Universal Robots PolyScope program: Cobot_soudure_29112023.urp

Program Cobot_soudure_29112023 (installation=Cobot_soudure_29112023 directory=/home/ur/ursim/ursim-5.11.0.108249/programs/TRAVAIL 27112023 createdIn=5.9.4.1031232 lastSavedIn=5.11.0.108249 robotSerialNumber=20195299999)
Calibrated DH parameters: a=[0, -0.6127, -0.57155, 0, 0, 0]; d=[0.1807, 0, 0, 0.17415, 0.11985, 0.11655]; alpha=[1.570796, 0, 0, 1.570796, -1.570796, 0]; deltaTheta=[0, 0, 0, 0, 0, 0]
InitVariablesNode variables(variable(name=Test_Gaz, expression=False), variable(name=Test_Job, expression=False), variable(name=Test_Ordre_Mar, expression=False), variable(name=Valide_Gaz, expression=False), variable(name=fin_soud, expression=1), variable(name=secu_d, expression=0), variable(name=secu_g, expression=0), variable(name=timer_ret_gaz, expression=0))
BeforeStart
  Folder fonctions
    Folder Init [hidden by the author, left out]
    Folder Diverses
      Script file /home/ur/ursim/ursim-5.11.0.108249/programs/SCRIPT/Scripts_soudure/Diverses/close_popup.script
        | #fermeture popup
        | 
        | def close_popup():
        | 	closepop = "close popup"
        |     	socket_send_string(closepop,"internal")
        |     	socket_send_byte(10,"internal")
        |     	socket_close()
        | 
        | 	closepop = "close popup"
        |     	socket_send_string(closepop,"internal")
        |     	socket_send_byte(10,"internal")
        |     	socket_close()
        | 	return(False)
        | end
      Script file /home/ur/ursim/ursim-5.11.0.108249/programs/SCRIPT/Scripts_soudure/Diverses/debut_soud.script
        | def fun_debut_soudure():
        |     Valide_Gaz = False
        |     if  ((Test_Ordre_Mar == False) and (Test_Job == False)):
        |         Arc_On = True
        |         Test_Gaz = True
        |     end
        | end
      Script file /home/ur/ursim/ursim-5.11.0.108249/programs/SCRIPT/Scripts_soudure/Diverses/fin_soudure.script
        | def fin_soudure():
        |         Arc_On = False
        |         Test_Gaz = False
        |         Test_Job = True
        |         Test_Ordre_Mar = True
        | end
      Script file /home/ur/ursim/ursim-5.11.0.108249/programs/SCRIPT/Scripts_soudure/Diverses/fun_demande_job.script
        | #demande le job à utiliser (mode de soudure régler sur le poste à souder) (compris entre 0 et 3, pour 1 et 4 sur le poste a souder)
        | def fun_demande_job(type):
        | 	if (1==type):
        | 		soudure = "point"
        | 	elif (2==type):
        | 		soudure = "lineaire"
        | 	elif (3==type):
        | 		soudure = "arc de cercle"
        | 	elif (4==type):
        | 		soudure = "cercle"
        | 	elif (5==type):
        | 		soudure = "lineaire + balayage"
        | 	elif (6==type):
        | 		soudure = "Recopie"
        | 	else :
        | 		return(False)
        | 	end
        | 
        |   job = request_integer_from_primary_client("Mode du poste à souder pour soudure : "+ soudure + " ? [1-4]")
        |   #job = job-1 #adapter la saisie aux besoins du code
        | 
        |   while ((job!=4) and (job!=1) and (job!=2) and (job!=3)): #reboucler si mauvaise saisie
        | 	  job = request_integer_from_primary_client("Mode du poste à souder pour soudure : "+ soudure + " ? [1-4]")
        |       #job = job-1 #adapter la saisie aux besoins du code
        |   end
        | 
        | return(job)
        | end
      Script file /home/ur/ursim/ursim-5.11.0.108249/programs/SCRIPT/Scripts_soudure/Diverses/fun_demande_type_soudure.script
        | #demande le type de soudure à enregistrer (entre 1 et 5)
        | def fun_demande_type_soudure():
        |     sync()
        | 	reponse = request_integer_from_primary_client("1->POINT     2->LINEAIRE    3->ARC    4->CERCLE  5->LINEAIRE BALAYAGE     6->RECOPIE     7->FIN")
        |     sync()
        |     if ((reponse == 0) or (reponse >= 7)):
        |         reponse = 7
        |     end
        |     sync()
        | return(reponse)
        | end
      SuppressedNode
        Script file /home/ur/ursim/ursim-5.11.0.108249/programs/SCRIPT/Scripts_soudure/Diverses/fun_demande().script
          | #demande nombre soudures par type (compris entre 0 et 6)
          | 
          | def fun_demande(type):
          | 	if (1==type):
          | 		soudure = "point"					#si type = 1, la demande sera sur une soudure point
          | 	elif (2==type):
          | 		soudure = "lineaire"				#si type = 2, la demande sera sur une soudure linéaire
          | 	elif (3==type):
          | 		soudure = "arc de cercle"			#si type = 3, la demande sera sur une soudure arc de cercle
          | 	elif (4==type):
          | 		soudure = "cercle"					#si type = 4, la demande sera sur une soudure cercle
          | 	elif (5==type):
          | 		soudure = "lineaire + balayage"
          | 	else :
          | 		return(False)
          | 	end
          | 
          | 	nb_soud = request_integer_from_primary_client("nombre de soudure(s) "+ soudure + " ?")			#la demande
          | 	if (nb_soud >6):																									#si la reponse est superieur a 6
          | 		popup1 = "popup le robot ne peut pas effectuer plus de 6 soudures "+ soudure + " sur la même pièce, réessayer."	#popup
          | 		socket_open("127.0.0.1",29999,"internal") # open internal socket
          | 
          | 		socket_send_line(popup1,"internal")         #Affichage Popup
          | 
          | 		socket_send_byte(10,"internal")
          | 		sleep(5.0)
          | 		closepop = "close popup"					#fermer popup
          | 		socket_send_string(closepop,"internal")
          | 		socket_send_byte(10,"internal")
          | 		socket_close()
          | 
          | 		while(nb_soud >6):
          | 			nb_soud = request_integer_from_primary_client("nombre de soudure(s) "+ soudure + " ? (compris entre 0 et 6 ;)")	#on redemande tant que le nombre est superieur a 6
          | 		end
          | end
          | return(nb_soud)        #on retourne le nombre de soudure à effectuer dans le type
          | end
      Script file /home/ur/ursim/ursim-5.11.0.108249/programs/SCRIPT/Scripts_soudure/Diverses/fun_demande_vit.script
        | #demande nombre soudures par type (compris entre 0 et 6)
        | def fun_demande_vit(type):
        | 	if (1==type):
        | 		soudure = "point"
        | 	elif (2==type):
        | 		soudure = "lineaire"
        | 	elif (3==type):
        | 		soudure = "arc de cercle"
        | 	elif (4==type):
        | 		soudure = "cercle"
        | 	else :
        | 		return(False)
        | 	end
        | 
        | vit_soud = request_float_from_primary_client("vitesse de la soudure "+ soudure + " ? (mm/s)")
        | 	#if (vit_soud >6):
        | 	#	popup1 = "popup le robot ne peut pas effectuer plus de 6 soudures "+ soudure + " sur la même pièce, réessayer."
        | 	#	socket_open("127.0.0.1",29999,"internal") # open internal socket
        | 
        | 	#	socket_send_line(popup1,"internal")         #Affichage Popup
        | 
        | 	#	socket_send_byte(10,"internal")
        | 	#	sleep(5.0)
        | 	#	closepop = "close popup"
        | 	#	socket_send_string(closepop,"internal")
        | 	#	socket_send_byte(10,"internal")
        | 	#	socket_close()
        | 
        | 	#	while(vit_soud >6):
        | 	#		vit_soud = request_integer_from_primary_client("nombre de soudure(s) "+ soudure + " ? (compris entre 0 et 6 ;)")
        | 	#	end
        | #end
        | return(vit_soud/1000)
        | end
      Script file /home/ur/ursim/ursim-5.11.0.108249/programs/SCRIPT/Scripts_soudure/Diverses/fun_front_down.script
        | #attente front montant sur add_bp
        | 
        | def fun_front_do(add_bp):
        | bp = get_digital_in(add_bp)
        |     while not bp :
        |         bp = get_digital_in(add_bp)    #dans la boucle tant que l'entrée add_bp est a 1
        |         #attente relachement bouton
        |    end
        | 
        |     while bp :                              #dans la boucle tant que l'entrée add_bp est a 0
        |         bp = get_digital_in(add_bp)
        |         #attente
        |     end
        | 
        |     #while not bp :
        |            #bp = get_digital_in(add_bp)    #dans la boucle tant que l'entrée add_bp est a 1
        |      #end
        | 
        |     return(False)
        | end
      Script file /home/ur/ursim/ursim-5.11.0.108249/programs/SCRIPT/Scripts_soudure/Diverses/fun_front_up.script
        | #attente front montant sur add_bp
        | 
        | def fun_front_up(add_bp):
        | bp = get_digital_in(add_bp)
        |     while bp :
        |         bp = get_digital_in(add_bp)    #dans la boucle tant que l'entrée add_bp est a 14
        |         sync()
        |         #attente relachement bouton
        |     end
        |     sync()
        |     while not bp :                              #dans la boucle tant que l'entrée add_bp est a 0
        |         bp = get_digital_in(add_bp)
        |         sync()
        |         #attente
        |     end
        |     sync()
        |     return(False)
        | end
      Script file /home/ur/ursim/ursim-5.11.0.108249/programs/SCRIPT/Scripts_soudure/Diverses/fun_popup_soud().script
        | #ouvre un pop-up "configuration soudure (type_soud) n°(num_soud): placer le robot (etape_soud) et valider la position. (bp_cobot)". fermeture popup a l'aide de close_popup()
        | #pour la definition de la fonction :
        |     #etape :
        |     #   1 : approche
        |     #   2 : depart
        |     #   3 : premier quart
        |     #   4 : milieu
        |     #   5 : trois-quart
        |     #   6 : fin
        |     #   7 : retrait
        | 
        |     #type :
        |     #   1 : soudure point
        |     #   2 : soudure lineaire
        |     #   3 : soudure arc de cercle
        |     #   4 : soudure cercle
        |     #   5 : plus de soudure
        |     #num : i, j, k ou l correspondant au numero de la soudure ( i pour type = 1, j pour type = 2, k pour type = 3, l pour type = 4)
        | 
        | def fun_popup_soud(etape, type, num):
        |     sync()
        |     switch_1 = etape
        |     switch_2 = type
        |         ##############################################################################
        | 
        |     ####################### POPUP-approche #######################################
        | 
        | ##############################################################################
        |     #switch etape
        |     if (1 == switch_1) : #point d'approche
        |         etape_soud = " en APPROCHE"
        |         #switch type
        |         if (1 == switch_2) : #soudure point
        |             type_soud = "point"
        | 
        |        elif (2 == switch_2) : #soudure lineaire
        |             type_soud = "lineaire"
        | 
        |         elif (3 == switch_2) : #soudure arc de cerlce
        |             type_soud = "arc de cercle"
        | 
        |         elif (4 == switch_2) : #soudure cercle
        |            type_soud = "cercle"
        | 
        |         else :
        |             return (False)
        |         end
        | 
        |         ##############################################################################
        | 
        |     ####################### POPUP-debut ##########################################
        | 
        | ##############################################################################
        | 
        |     elif (2 == switch_1): #point de soudure/debut
        |         #switch type
        |         if (1 == switch_2) : #soudure point
        |            etape_soud = "sur le POINT"
        |             type_soud = "point"
        | 
        |         elif (2 == switch_2): #soudure lineaire
        |             etape_soud = "sur le DEBUT"
        |             type_soud = "lineaire"
        | 
        |         elif (3 == switch_2) : #soudure arc de cerlce
        |             etape_soud = "sur le DEBUT"
        |             type_soud = "arc de cercle"
        | 
        |         elif (4 == switch_2) : #soudure cercle
        |             etape_soud = "sur le DEBUT"
        |            type_soud = "cercle"
        | 
        |         else :
        |             return (False)
        |         end
        | 
        |         ##############################################################################
        | 
        |     ####################### POPUP-quart ##########################################
        | 
        | ##############################################################################
        | 
        |     elif (3 == switch_1): #point de quart
        |         etape_soud = "sur 1er QUART"
        |         #switch type
        |         if (4 == switch_2) : #soudure cercle
        |             type_soud = "cercle"
        |         end
        | 
        |         ##############################################################################
        | 
        |     ####################### POPUP-milieu ########################################
        | 
        | #############################################################################
        | 
        |     elif (4 == switch_1): #point de milieu
        |         etape_soud = "à la MOITIE"
        |         #switch type
        |         if (3 == switch_2) : #soudure arc de cercle
        |             type_soud = "arc de cercle"
        |         elif (4 == switch_2): #soudure arc de cercle
        |             type_soud = "cercle"
        |         end
        | 
        |         ##############################################################################
        | 
        |     ####################### POPUP-trois_quart ####################################
        | 
        | ##############################################################################
        | 
        |     elif (5 == switch_1): #point trois_quart
        |         etape_soud = "sur le 3e QUART"
        |         #switch type
        |         if (4 == switch_2) : #soudure cercle
        |             type_soud = "cercle"
        |         end
        | 
        |         ##############################################################################
        | 
        |     ####################### POPUP-fin ############################################
        | 
        | ##############################################################################
        | 
        |     elif (6 == switch_1): #point de fin
        |         etape_soud = "sur la FIN"
        |         #switch type
        |         if (2 == switch_2) : #soudure lineaire
        |             type_soud = "lineaire"
        | 
        |         elif (3 == switch_2) : #soudure arc de cerlce
        |             type_soud = "arc de cercle"
        | 
        |         elif (4 == switch_2) : #soudure cercle
        |             type_soud = "cercle"
        | 
        |         else :
        |             return (False)
        |         end
        | 
        |         ##############################################################################
        | 
        |     ####################### POPUP-retrait ########################################
        | 
        | ##############################################################################
        | 
        |     elif (7 == switch_1): #point de retrait
        |         etape_soud = "en RETRAIT"
        |         #switch type
        |         if (2 == switch_2) : #soudure lineaire
        |             type_soud = "lineaire"
        | 
        |         elif (3 == switch_2) : #soudure arc de cerlce
        |            type_soud = "arc de cercle"
        | 
        |         elif (4 == switch_2) : #soudure cercle
        |            type_soud = "cercle"
        | 
        |         else :
        |            return (False)
        |         end
        | 
        |     else :
        |         return(False)
        |     end
        | 
        |         ##############################################################################
        | 
        |     ######################## affichage_POPUP #####################################
        | 
        | ##############################################################################
        |     sync()
        |     num_soud = to_str(num)
        |     popup1 = "popup Config. : " + type_soud + " n°" + num_soud + " : placer " + etape_soud + " & Valider"             #on ouvre un popup
        |     socket_open("127.0.0.1",29999,"internal") # open internal socket
        |     socket_send_line(popup1,"internal")     #Affichage message
        |     socket_send_byte(10,"internal")
        |     sync()
        | end
      Script file /home/ur/ursim/ursim-5.11.0.108249/programs/SCRIPT/Scripts_soudure/Diverses/fun_raz_d.script
        | def fun_raz_d():
        |     #taille des tableaux de positions = nombre de soudures maximum par type + 1 (car commence à enregistrer à l'index 1)
        |     global tab_point_app_d =    [p[0,0,0,0,0,0], p[0,0,0,0,0,0], p[0,0,0,0,0,0], p[0,0,0,0,0,0], p[0,0,0,0,0,0], p[0,0,0,0,0,0], p[0,0,0,0,0,0], p[0,0,0,0,0,0], p[0,0,0,0,0,0], p[0,0,0,0,0,0], p[0,0,0,0,0,0]]
        |     global tab_point_deb_d =    [p[0,0,0,0,0,0], p[0,0,0,0,0,0], p[0,0,0,0,0,0], p[0,0,0,0,0,0], p[0,0,0,0,0,0], p[0,0,0,0,0,0], p[0,0,0,0,0,0], p[0,0,0,0,0,0], p[0,0,0,0,0,0], p[0,0,0,0,0,0], p[0,0,0,0,0,0]]
        |     global tab_point_ret_d =    [p[0,0,0,0,0,0], p[0,0,0,0,0,0], p[0,0,0,0,0,0], p[0,0,0,0,0,0], p[0,0,0,0,0,0], p[0,0,0,0,0,0], p[0,0,0,0,0,0], p[0,0,0,0,0,0], p[0,0,0,0,0,0], p[0,0,0,0,0,0], p[0,0,0,0,0,0]]
        | 
        |     global tab_lin_app_d =      [p[0,0,0,0,0,0], p[0,0,0,0,0,0], p[0,0,0,0,0,0], p[0,0,0,0,0,0], p[0,0,0,0,0,0], p[0,0,0,0,0,0], p[0,0,0,0,0,0], p[0,0,0,0,0,0], p[0,0,0,0,0,0], p[0,0,0,0,0,0], p[0,0,0,0,0,0]]
        |     global tab_lin_deb_d =      [p[0,0,0,0,0,0], p[0,0,0,0,0,0], p[0,0,0,0,0,0], p[0,0,0,0,0,0], p[0,0,0,0,0,0], p[0,0,0,0,0,0], p[0,0,0,0,0,0], p[0,0,0,0,0,0], p[0,0,0,0,0,0], p[0,0,0,0,0,0], p[0,0,0,0,0,0]]
        |     global tab_lin_fin_d =      [p[0,0,0,0,0,0], p[0,0,0,0,0,0], p[0,0,0,0,0,0], p[0,0,0,0,0,0], p[0,0,0,0,0,0], p[0,0,0,0,0,0], p[0,0,0,0,0,0], p[0,0,0,0,0,0], p[0,0,0,0,0,0], p[0,0,0,0,0,0], p[0,0,0,0,0,0]]
        |     global tab_lin_ret_d =      [p[0,0,0,0,0,0], p[0,0,0,0,0,0], p[0,0,0,0,0,0], p[0,0,0,0,0,0], p[0,0,0,0,0,0], p[0,0,0,0,0,0], p[0,0,0,0,0,0], p[0,0,0,0,0,0], p[0,0,0,0,0,0], p[0,0,0,0,0,0], p[0,0,0,0,0,0]]
        | 
        |     global tab_arc_app_d =      [p[0,0,0,0,0,0], p[0,0,0,0,0,0], p[0,0,0,0,0,0], p[0,0,0,0,0,0], p[0,0,0,0,0,0], p[0,0,0,0,0,0], p[0,0,0,0,0,0], p[0,0,0,0,0,0], p[0,0,0,0,0,0], p[0,0,0,0,0,0], p[0,0,0,0,0,0]]
        |     global tab_arc_deb_d =      [p[0,0,0,0,0,0], p[0,0,0,0,0,0], p[0,0,0,0,0,0], p[0,0,0,0,0,0], p[0,0,0,0,0,0], p[0,0,0,0,0,0], p[0,0,0,0,0,0], p[0,0,0,0,0,0], p[0,0,0,0,0,0], p[0,0,0,0,0,0], p[0,0,0,0,0,0]]
        |     global tab_arc_mil_d =      [p[0,0,0,0,0,0], p[0,0,0,0,0,0], p[0,0,0,0,0,0], p[0,0,0,0,0,0], p[0,0,0,0,0,0], p[0,0,0,0,0,0], p[0,0,0,0,0,0], p[0,0,0,0,0,0], p[0,0,0,0,0,0], p[0,0,0,0,0,0], p[0,0,0,0,0,0]]
        |     global tab_arc_fin_d =      [p[0,0,0,0,0,0], p[0,0,0,0,0,0], p[0,0,0,0,0,0], p[0,0,0,0,0,0], p[0,0,0,0,0,0], p[0,0,0,0,0,0], p[0,0,0,0,0,0], p[0,0,0,0,0,0], p[0,0,0,0,0,0], p[0,0,0,0,0,0], p[0,0,0,0,0,0]]
        |     global tab_arc_ret_d =      [p[0,0,0,0,0,0], p[0,0,0,0,0,0], p[0,0,0,0,0,0], p[0,0,0,0,0,0], p[0,0,0,0,0,0], p[0,0,0,0,0,0], p[0,0,0,0,0,0], p[0,0,0,0,0,0], p[0,0,0,0,0,0], p[0,0,0,0,0,0], p[0,0,0,0,0,0]]
        | 
        |     global tab_cer_app_d =      [p[0,0,0,0,0,0], p[0,0,0,0,0,0], p[0,0,0,0,0,0], p[0,0,0,0,0,0], p[0,0,0,0,0,0], p[0,0,0,0,0,0], p[0,0,0,0,0,0], p[0,0,0,0,0,0], p[0,0,0,0,0,0], p[0,0,0,0,0,0], p[0,0,0,0,0,0]]
        |     global tab_cer_deb_d =      [p[0,0,0,0,0,0], p[0,0,0,0,0,0], p[0,0,0,0,0,0], p[0,0,0,0,0,0], p[0,0,0,0,0,0], p[0,0,0,0,0,0], p[0,0,0,0,0,0], p[0,0,0,0,0,0], p[0,0,0,0,0,0], p[0,0,0,0,0,0], p[0,0,0,0,0,0]]
        |     global tab_cer_quart_d =    [p[0,0,0,0,0,0], p[0,0,0,0,0,0], p[0,0,0,0,0,0], p[0,0,0,0,0,0], p[0,0,0,0,0,0], p[0,0,0,0,0,0], p[0,0,0,0,0,0], p[0,0,0,0,0,0], p[0,0,0,0,0,0], p[0,0,0,0,0,0], p[0,0,0,0,0,0]]
        |     global tab_cer_mil_d =      [p[0,0,0,0,0,0], p[0,0,0,0,0,0], p[0,0,0,0,0,0], p[0,0,0,0,0,0], p[0,0,0,0,0,0], p[0,0,0,0,0,0], p[0,0,0,0,0,0], p[0,0,0,0,0,0], p[0,0,0,0,0,0], p[0,0,0,0,0,0], p[0,0,0,0,0,0]]
        |     global tab_cer_tro_d =      [p[0,0,0,0,0,0], p[0,0,0,0,0,0], p[0,0,0,0,0,0], p[0,0,0,0,0,0], p[0,0,0,0,0,0], p[0,0,0,0,0,0], p[0,0,0,0,0,0], p[0,0,0,0,0,0], p[0,0,0,0,0,0], p[0,0,0,0,0,0], p[0,0,0,0,0,0]]
        |     global tab_cer_fin_d =      [p[0,0,0,0,0,0], p[0,0,0,0,0,0], p[0,0,0,0,0,0], p[0,0,0,0,0,0], p[0,0,0,0,0,0], p[0,0,0,0,0,0], p[0,0,0,0,0,0], p[0,0,0,0,0,0], p[0,0,0,0,0,0], p[0,0,0,0,0,0], p[0,0,0,0,0,0]]
        |     global tab_cer_ret_d =      [p[0,0,0,0,0,0], p[0,0,0,0,0,0], p[0,0,0,0,0,0], p[0,0,0,0,0,0], p[0,0,0,0,0,0], p[0,0,0,0,0,0], p[0,0,0,0,0,0], p[0,0,0,0,0,0], p[0,0,0,0,0,0], p[0,0,0,0,0,0], p[0,0,0,0,0,0]]
        | 
        |      #2 nouveaux tableaux modif V2.1 (longueur 40 si 4(type)*10(nb soudures max par type) ) -> mis 45 (permettre décalage + marge)
        |     global tab_type_d = [0,0,0,0,0,0,0,0,0,0,0,0,0,0,0,0,0,0,0,0,0,0,0,0,0,0,0,0,0,0,0,0,0,0,0,0,0,0,0,0,0,0,0,0,0]
        |     global tab_job_d  = [0,0,0,0,0,0,0,0,0,0,0,0,0,0,0,0,0,0,0,0,0,0,0,0,0,0,0,0,0,0,0,0,0,0,0,0,0,0,0,0,0,0,0,0,0]
        | 
        |     #vitesses de soudure
        |     global tps_point_d = 0
        |     global vit_arc_d = [0,0,0,0,0,0,0,0,0,0,0]
        |     global vit_cer_d = [0,0,0,0,0,0,0,0,0,0,0]
        |     global vit_lin_d = [0,0,0,0,0,0,0,0,0,0,0]
        | 
        |     global nb_soud_point_d  = 0
        |     global nb_soud_lin_d    = 0
        |     global nb_soud_arc_d    = 0
        |     global nb_soud_cer_d    = 0
        | 
        |     global nbSoudure_glo_d  = 0
        | 
        | end
      Script file /home/ur/ursim/ursim-5.11.0.108249/programs/SCRIPT/Scripts_soudure/Diverses/fun_raz_g.script
        | def fun_raz_g():
        |     #taille des tableaux de positions = nombre de soudures maximum par type + 1 (car commence à enregistrer à l'index 1)
        |     global tab_point_app_g =    [p[0,0,0,0,0,0], p[0,0,0,0,0,0], p[0,0,0,0,0,0], p[0,0,0,0,0,0], p[0,0,0,0,0,0], p[0,0,0,0,0,0], p[0,0,0,0,0,0], p[0,0,0,0,0,0], p[0,0,0,0,0,0], p[0,0,0,0,0,0], p[0,0,0,0,0,0]]
        |     global tab_point_deb_g =    [p[0,0,0,0,0,0], p[0,0,0,0,0,0], p[0,0,0,0,0,0], p[0,0,0,0,0,0], p[0,0,0,0,0,0], p[0,0,0,0,0,0], p[0,0,0,0,0,0], p[0,0,0,0,0,0], p[0,0,0,0,0,0], p[0,0,0,0,0,0], p[0,0,0,0,0,0]]
        |     global tab_point_ret_g =    [p[0,0,0,0,0,0], p[0,0,0,0,0,0], p[0,0,0,0,0,0], p[0,0,0,0,0,0], p[0,0,0,0,0,0], p[0,0,0,0,0,0], p[0,0,0,0,0,0], p[0,0,0,0,0,0], p[0,0,0,0,0,0], p[0,0,0,0,0,0], p[0,0,0,0,0,0]]
        | 
        |     global tab_lin_app_g =      [p[0,0,0,0,0,0], p[0,0,0,0,0,0], p[0,0,0,0,0,0], p[0,0,0,0,0,0], p[0,0,0,0,0,0], p[0,0,0,0,0,0], p[0,0,0,0,0,0], p[0,0,0,0,0,0], p[0,0,0,0,0,0], p[0,0,0,0,0,0], p[0,0,0,0,0,0]]
        |     global tab_lin_deb_g =      [p[0,0,0,0,0,0], p[0,0,0,0,0,0], p[0,0,0,0,0,0], p[0,0,0,0,0,0], p[0,0,0,0,0,0], p[0,0,0,0,0,0], p[0,0,0,0,0,0], p[0,0,0,0,0,0], p[0,0,0,0,0,0], p[0,0,0,0,0,0], p[0,0,0,0,0,0]]
        |     global tab_lin_fin_g =      [p[0,0,0,0,0,0], p[0,0,0,0,0,0], p[0,0,0,0,0,0], p[0,0,0,0,0,0], p[0,0,0,0,0,0], p[0,0,0,0,0,0], p[0,0,0,0,0,0], p[0,0,0,0,0,0], p[0,0,0,0,0,0], p[0,0,0,0,0,0], p[0,0,0,0,0,0]]
        |     global tab_lin_ret_g =      [p[0,0,0,0,0,0], p[0,0,0,0,0,0], p[0,0,0,0,0,0], p[0,0,0,0,0,0], p[0,0,0,0,0,0], p[0,0,0,0,0,0], p[0,0,0,0,0,0], p[0,0,0,0,0,0], p[0,0,0,0,0,0], p[0,0,0,0,0,0], p[0,0,0,0,0,0]]
        | 
        |     global tab_arc_app_g =      [p[0,0,0,0,0,0], p[0,0,0,0,0,0], p[0,0,0,0,0,0], p[0,0,0,0,0,0], p[0,0,0,0,0,0], p[0,0,0,0,0,0], p[0,0,0,0,0,0], p[0,0,0,0,0,0], p[0,0,0,0,0,0], p[0,0,0,0,0,0], p[0,0,0,0,0,0]]
        |     global tab_arc_deb_g =      [p[0,0,0,0,0,0], p[0,0,0,0,0,0], p[0,0,0,0,0,0], p[0,0,0,0,0,0], p[0,0,0,0,0,0], p[0,0,0,0,0,0], p[0,0,0,0,0,0], p[0,0,0,0,0,0], p[0,0,0,0,0,0], p[0,0,0,0,0,0], p[0,0,0,0,0,0]]
        |     global tab_arc_mil_g =      [p[0,0,0,0,0,0], p[0,0,0,0,0,0], p[0,0,0,0,0,0], p[0,0,0,0,0,0], p[0,0,0,0,0,0], p[0,0,0,0,0,0], p[0,0,0,0,0,0], p[0,0,0,0,0,0], p[0,0,0,0,0,0], p[0,0,0,0,0,0], p[0,0,0,0,0,0]]
        |     global tab_arc_fin_g =      [p[0,0,0,0,0,0], p[0,0,0,0,0,0], p[0,0,0,0,0,0], p[0,0,0,0,0,0], p[0,0,0,0,0,0], p[0,0,0,0,0,0], p[0,0,0,0,0,0], p[0,0,0,0,0,0], p[0,0,0,0,0,0], p[0,0,0,0,0,0], p[0,0,0,0,0,0]]
        |     global tab_arc_ret_g =      [p[0,0,0,0,0,0], p[0,0,0,0,0,0], p[0,0,0,0,0,0], p[0,0,0,0,0,0], p[0,0,0,0,0,0], p[0,0,0,0,0,0], p[0,0,0,0,0,0], p[0,0,0,0,0,0], p[0,0,0,0,0,0], p[0,0,0,0,0,0], p[0,0,0,0,0,0]]
        | 
        |     global tab_cer_app_g =      [p[0,0,0,0,0,0], p[0,0,0,0,0,0], p[0,0,0,0,0,0], p[0,0,0,0,0,0], p[0,0,0,0,0,0], p[0,0,0,0,0,0], p[0,0,0,0,0,0], p[0,0,0,0,0,0], p[0,0,0,0,0,0], p[0,0,0,0,0,0], p[0,0,0,0,0,0]]
        |     global tab_cer_deb_g =      [p[0,0,0,0,0,0], p[0,0,0,0,0,0], p[0,0,0,0,0,0], p[0,0,0,0,0,0], p[0,0,0,0,0,0], p[0,0,0,0,0,0], p[0,0,0,0,0,0], p[0,0,0,0,0,0], p[0,0,0,0,0,0], p[0,0,0,0,0,0], p[0,0,0,0,0,0]]
        |     global tab_cer_quart_g =    [p[0,0,0,0,0,0], p[0,0,0,0,0,0], p[0,0,0,0,0,0], p[0,0,0,0,0,0], p[0,0,0,0,0,0], p[0,0,0,0,0,0], p[0,0,0,0,0,0], p[0,0,0,0,0,0], p[0,0,0,0,0,0], p[0,0,0,0,0,0], p[0,0,0,0,0,0]]
        |     global tab_cer_mil_g =      [p[0,0,0,0,0,0], p[0,0,0,0,0,0], p[0,0,0,0,0,0], p[0,0,0,0,0,0], p[0,0,0,0,0,0], p[0,0,0,0,0,0], p[0,0,0,0,0,0], p[0,0,0,0,0,0], p[0,0,0,0,0,0], p[0,0,0,0,0,0], p[0,0,0,0,0,0]]
        |     global tab_cer_tro_g =      [p[0,0,0,0,0,0], p[0,0,0,0,0,0], p[0,0,0,0,0,0], p[0,0,0,0,0,0], p[0,0,0,0,0,0], p[0,0,0,0,0,0], p[0,0,0,0,0,0], p[0,0,0,0,0,0], p[0,0,0,0,0,0], p[0,0,0,0,0,0], p[0,0,0,0,0,0]]
        |     global tab_cer_fin_g =      [p[0,0,0,0,0,0], p[0,0,0,0,0,0], p[0,0,0,0,0,0], p[0,0,0,0,0,0], p[0,0,0,0,0,0], p[0,0,0,0,0,0], p[0,0,0,0,0,0], p[0,0,0,0,0,0], p[0,0,0,0,0,0], p[0,0,0,0,0,0], p[0,0,0,0,0,0]]
        |     global tab_cer_ret_g =      [p[0,0,0,0,0,0], p[0,0,0,0,0,0], p[0,0,0,0,0,0], p[0,0,0,0,0,0], p[0,0,0,0,0,0], p[0,0,0,0,0,0], p[0,0,0,0,0,0], p[0,0,0,0,0,0], p[0,0,0,0,0,0], p[0,0,0,0,0,0], p[0,0,0,0,0,0]]
        | 
        |      #2 nouveaux tableaux modif V2.1 (longueur 40 si 4(type)*10(nb soudures max par type) ) -> mis 45 (permettre décalage + marge)
        |     global tab_type_g = [0,0,0,0,0,0,0,0,0,0,0,0,0,0,0,0,0,0,0,0,0,0,0,0,0,0,0,0,0,0,0,0,0,0,0,0,0,0,0,0,0,0,0,0,0]
        |     global tab_job_g  = [0,0,0,0,0,0,0,0,0,0,0,0,0,0,0,0,0,0,0,0,0,0,0,0,0,0,0,0,0,0,0,0,0,0,0,0,0,0,0,0,0,0,0,0,0]
        | 
        |     #vitesses de soudure
        |     global tps_point_g = 0
        |     global vit_arc_g = [0,0,0,0,0,0,0,0,0,0,0]
        |     global vit_cer_g = [0,0,0,0,0,0,0,0,0,0,0]
        |     global vit_lin_g = [0,0,0,0,0,0,0,0,0,0,0]
        | 
        |     global nb_soud_point_g  = 0
        |     global nb_soud_lin_g    = 0
        |     global nb_soud_arc_g    = 0
        |     global nb_soud_cer_g    = 0
        | 
        |     global nbSoudure_glo_g  = 0
        | end
    SuppressedNode
      Folder Demande [hidden by the author, left out]
    Folder Configuration [hidden by the author, left out]
    Folder Execution [hidden by the author, left out]
    Folder Pas_A_Pas [hidden by the author, left out]
    Folder PopUps [hidden by the author, left out]
    Folder Mouvements soudures [hidden by the author, left out]
    Folder General [hidden by the author, left out]
Robot Program (runOnlyOnce=true)
  Script: General()
SubProgram Recopie_Table_Droite [hidden by the author, left out]
SubProgram Recopie_Table_Gauche [hidden by the author, left out]
Thread Thread_1 (runOnlyOnce=false)
  Folder Test_Ordre_Marche [hidden by the author, left out]
  Script: sync()
Thread Thread_2 (runOnlyOnce=false)
  Folder mode_soudure [hidden by the author, left out]
  Script: sync()
Thread Thread_3 (runOnlyOnce=false)
  Folder led_cobot_2 [hidden by the author, left out]
  Script: sync()
Thread Thread_4 (runOnlyOnce=false)
  Folder led_cobot [hidden by the author, left out]
  Script: sync()
Thread Thread_5 (runOnlyOnce=false)
  Folder Test_Arc_On [hidden by the author, left out]
  Script: sync()
SuppressedNode
  Thread Thread_6 (runOnlyOnce=false)
    Folder Test_Job
      If Test_Job≟ True
        SuppressedNode
          If Program_Soudure≟1 removedSiblings(If(type=ElseIf checkContinuously=false, expression=Program_Soudure≟2, children(Set(type=DigitalOutput, pin=Job_1, digitalValue=0), Set(type=DigitalOutput, pin=Job_2, digitalValue=1))), If(type=ElseIf checkContinuously=false, expression=Program_Soudure≟3, children(Set(type=DigitalOutput, pin=Job_1, digitalValue=1), Set(type=DigitalOutput, pin=Job_2, digitalValue=1))), If(type=ElseIf checkContinuously=false, expression=Program_Soudure≟4, children(Set(type=DigitalOutput, pin=Job_1, digitalValue=0), Set(type=DigitalOutput, pin=Job_2, digitalValue=0))), If(type=Else checkContinuously=false, children(Script(type=Line, expression=close_popup()), Popup(type=Error haltProgram=false message=Le Job soudure choisi n'existe pas. inputType=Text))))
            Set DigitalOutput pin=Job_1; digitalValue=1
            Set DigitalOutput pin=Job_2; digitalValue=0
        Test_Job := False
    Script: sync()
Thread Thread_7 (runOnlyOnce=false)
  Folder secu [hidden by the author, left out]
  Script: sync()
Thread Thread_8 (runOnlyOnce=false)
  Folder bloq_soud_arret [hidden by the author, left out]
  SuppressedNode
    Folder freedrive_droit
      If led_cobot ≟  True
        If tool_in[1] ≟ True
          Script: teach_mode()
        Else 
          Script: end_teach_mode()
  Script: sync()
SuppressedNode
  Thread Thread_9 (runOnlyOnce=false)
    Folder reglage
      If reglage_d ≠0
        Script file /programs/Programmes/cobot_v2/sript/Part_reglage/REGLAGE_D.script
          |     ##############################################################################
          | 
          | ########################soudure point#########################################
          | 
          |     ##############################################################################
          | 
          |         if reglage_d == 1:                                    #remplissage tableau
          |             teach_mode()
          |             fun_popup_soud(1, 1, i)
          |             fun_front_up(adresse_bp_cobot)
          |             tab_point_app_d[i] =  get_actual_tcp_pose()     #Enregistrer position dans tableau d'approche des soudue points quand appui bouton
          |             close_popup()
          | 
          |             fun_popup_soud(2, 1, i)
          |             fun_front_up(adresse_bp_cobot)
          |             tab_point_deb_d[i] =  get_actual_tcp_pose()     #Enregistrer position debut quand appui bouton bp_cobot
          |             close_popup()
          | 
          |             tab_point_ret_d[i] = tab_point_app_d[i]         #point de retrait est le meme que le point d approche
          |             end_teach_mode()
          |             global reconfig = 1
          |             global reglage_d = 0
          | 
          |             sync()
          | 
          |         ##############################################################################
          | 
          |     ##############################################################################
          | 
          | ########################soudure lineaire######################################
          | 
          |     ##############################################################################
          | 
          |         elif reglage_d == 2:                		            #remplissage tableau
          |             teach_mode()
          |             fun_popup_soud(1, 2, j)
          |             fun_front_up(adresse_bp_cobot)
          |             tab_lin_app_d[j] =  get_actual_tcp_pose()     	#Enregistrer position dans tableau d approche des soudures lineaire quand appui Bp_cobot
          |             close_popup()
          | 
          |             fun_popup_soud(2, 2, j)
          |             fun_front_up(adresse_bp_cobot)
          |             tab_lin_deb_d[j] =  get_actual_tcp_pose()     	#Enregistrer position dans tableau debut quand appui Bp_cobot
          |             close_popup()
          | 
          |             fun_popup_soud(6, 2, j)
          |             fun_front_up(adresse_bp_cobot)
          |             tab_lin_fin_d[j] =  get_actual_tcp_pose()     	#Enregistrer position dans un tableau fin quand appui Bp_cobot
          |             close_popup()
          | 
          |             vit_lin_d[j] = fun_demande_vit(2)
          | 
          |             fun_popup_soud(7, 2, j)
          |             fun_front_up(adresse_bp_cobot)
          |             tab_lin_ret_d[j] =  get_actual_tcp_pose()     	#Enregistrer position dans tableau retrait quand appui Bp_cobot
          |             close_popup()
          |             end_teach_mode()
          |             global reglage_d = 0
          | 
          |             sync()
          | 
          |         ##############################################################################
          | 
          |     ##############################################################################
          | 
          | #########################soudure arc de cercle##################################
          | 
          |     #################################################################################
          | 
          |         elif reglage_d == 3:                                  #remplissage tableau
          |             teach_mode()
          |             fun_popup_soud(1, 3, k)
          |             fun_front_up(adresse_bp_cobot)
          |             tab_arc_app_d[k] =  get_actual_tcp_pose() 	    #Enregistrer position dans tableau d approche des soudures arc de cercle quand appui
          |             close_popup()
          | 
          |             fun_popup_soud(2, 3, k)
          |             fun_front_up(adresse_bp_cobot)
          |             tab_arc_deb_d[k] =  get_actual_tcp_pose() 	    #Enregistrer position dans tableau debut quand appui Bp_d
          |             close_popup()
          | 
          |             fun_popup_soud(4, 3, k)
          |             fun_front_up(adresse_bp_cobot)
          |             tab_arc_mil_d[k] =  get_actual_tcp_pose() 	    #Enregistrer position dans tableau milieu quand appui Bp_cobot
          |             close_popup()
          | 
          |             fun_popup_soud(6, 3, k)
          |             fun_front_up(adresse_bp_cobot)
          |             tab_arc_fin_d[k] =  get_actual_tcp_pose() 	    #Enregistrer position dans un tableau fin quand appui Bp_cobot
          |             close_popup()
          | 
          |             vit_arc_d[k] = fun_demande_vit(3)               #demande de vitesse des soudures lineaire
          | 
          |             fun_popup_soud(7, 3, k)
          |             fun_front_up(adresse_bp_cobot)
          |             tab_arc_ret_d[k] =  get_actual_tcp_pose() 	    #Enregistrer position dans tableau retrait quand appui Bp_cobot
          |             close_popup()
          |             end_teach_mode()
          |             global reglage_d = 0
          | 
          |             sync()
          | 
          |         ##############################################################################
          | 
          |     ##############################################################################
          | 
          | ############################soudure cercle####################################
          | 
          |     #################################################################################
          | 
          |         elif reglage_d == 4:                                  #remplissage tableau
          |             teach_mode()
          |             fun_popup_soud(1, 4, l)
          |             fun_front_up(adresse_bp_cobot)
          |             tab_cer_app_d[l] =  get_actual_tcp_pose()     	#Enregistrer position dans tableau d approche des soudures arc de cercle quand appui Bp_cobot
          |             close_popup()
          | 
          |             fun_popup_soud(2, 4, l)
          |             fun_front_up(adresse_bp_cobot)
          |             tab_cer_deb_d[l] =  get_actual_tcp_pose()     	#Enregistrer position dans tableau debut quand appui Bp_cobot
          |             close_popup()
          | 
          |             fun_popup_soud(3, 4, l)
          |             fun_front_up(adresse_bp_cobot)
          |             tab_cer_quart_d[l] =  get_actual_tcp_pose()   	#Enregistrer position dans tableau d'approche des soudures arc de cercle quand appui Bp_d
          |             close_popup()
          | 
          |             fun_popup_soud(4, 4, l)
          |             fun_front_up(adresse_bp_cobot)
          |             tab_cer_mil_d[l] =  get_actual_tcp_pose()     	#Enregistrer position dans tableau milieu quand appui Bp_cobot
          |             close_popup()
          | 
          |             fun_popup_soud(5, 4, l)
          |             fun_front_up(adresse_bp_cobot)
          |             tab_cer_tro_d[l] =  get_actual_tcp_pose()     	#Enregistrer position dans tableau milieu quand appui Bp_cobot
          |             close_popup()
          | 
          |             fun_popup_soud(6, 4, l)
          |             fun_front_up(adresse_bp_cobot)
          |             tab_cer_fin_d[l] =  get_actual_tcp_pose()     	#Enregistrer position dans un tableau fin quand appui Bp_cobot
          |             close_popup()
          | 
          |             vit_cer_d[l] = fun_demande_vit(4)
          | 
          |             fun_popup_soud(7, 4, l)
          |             fun_front_up(adresse_bp_cobot)
          |             tab_cer_ret_d[l] =  get_actual_tcp_pose()    	#position de retrait est la meme que position d approche
          |             close_popup()
          |             end_teach_mode()
          |             global reglage_d = 0
          |             sync()
          | 
          |         end
          | 
          |     ##############################################################################
          | 
          | ############################################################
        Script: sync()
      If reglage_g ≠0
        Script file /programs/usbdisk_0/COBOT/finish/reg/REGLAGE_G.script
          |     ##############################################################################
          | 
          | ########################soudure point#########################################
          | 
          |     ##############################################################################
          | 
          |         if reglage_g == 1:                                    #remplissage tableau
          |             teach_mode()
          |             fun_popup_soud(1, 1, i)
          |             fun_front_up(adresse_bp_cobot)
          |             tab_point_app_g[i] =  get_actual_tcp_pose()     #Enregistrer position dans tableau d'approche des soudue points quand appui bouton
          |             close_popup()
          | 
          |             fun_popup_soud(2, 1, i)
          |             fun_front_up(adresse_bp_cobot)
          |             tab_point_deb_g[i] =  get_actual_tcp_pose()     #Enregistrer position debut quand appui bouton bp_cobot
          |             close_popup()
          | 
          |             tab_point_ret_g[i] = tab_point_app_g[i]         #point de retrait est le meme que le point d approche
          |             end_teach_mode()
          |             global reconfig = 1
          |             global reglage_g = 0
          | 
          |             sync()
          | 
          |         ##############################################################################
          | 
          |     ##############################################################################
          | 
          | ########################soudure lineaire######################################
          | 
          |     ##############################################################################
          | 
          |         elif reglage_g == 2:                		            #remplissage tableau
          |             teach_mode()
          |             fun_popup_soud(1, 2, j)
          |             fun_front_up(adresse_bp_cobot)
          |             tab_lin_app_g[j] =  get_actual_tcp_pose()     	#Enregistrer position dans tableau d approche des soudures lineaire quand appui Bp_cobot
          |             close_popup()
          | 
          |             fun_popup_soud(2, 2, j)
          |             fun_front_up(adresse_bp_cobot)
          |             tab_lin_deb_g[j] =  get_actual_tcp_pose()     	#Enregistrer position dans tableau debut quand appui Bp_cobot
          |             close_popup()
          | 
          |             fun_popup_soud(6, 2, j)
          |             fun_front_up(adresse_bp_cobot)
          |             tab_lin_fin_g[j] =  get_actual_tcp_pose()     	#Enregistrer position dans un tableau fin quand appui Bp_cobot
          |             close_popup()
          | 
          |             vit_lin_g[j] = fun_demande_vit(2)
          | 
          |             fun_popup_soud(7, 2, j)
          |             fun_front_up(adresse_bp_cobot)
          |             tab_lin_ret_g[j] =  get_actual_tcp_pose()     	#Enregistrer position dans tableau retrait quand appui Bp_cobot
          |             close_popup()
          |             end_teach_mode()
          |             global reglage_g = 0
          | 
          |             sync()
          | 
          |         ##############################################################################
          | 
          |     ##############################################################################
          | 
          | #########################soudure arc de cercle##################################
          | 
          |     #################################################################################
          | 
          |         elif reglage_g == 3:                                  #remplissage tableau
          |             teach_mode()
          |             fun_popup_soud(1, 3, k)
          |             fun_front_up(adresse_bp_cobot)
          |             tab_arc_app_g[k] =  get_actual_tcp_pose() 	    #Enregistrer position dans tableau d approche des soudures arc de cercle quand appui
          |             close_popup()
          | 
          |             fun_popup_soud(2, 3, k)
          |             fun_front_up(adresse_bp_cobot)
          |             tab_arc_deb_g[k] =  get_actual_tcp_pose() 	    #Enregistrer position dans tableau debut quand appui BP_cobot
          |             close_popup()
          | 
          |             fun_popup_soud(4, 3, k)
          |             fun_front_up(adresse_bp_cobot)
          |             tab_arc_mil_g[k] =  get_actual_tcp_pose() 	    #Enregistrer position dans tableau milieu quand appui Bp_cobot
          |             close_popup()
          | 
          |             fun_popup_soud(6, 3, k)
          |             fun_front_up(adresse_bp_cobot)
          |             tab_arc_fin_g[k] =  get_actual_tcp_pose() 	    #Enregistrer position dans un tableau fin quand appui Bp_cobot
          |             close_popup()
          | 
          |             vit_arc_g[k] = fun_demande_vit(3)               #demande de vitesse des soudures lineaire
          | 
          |             fun_popup_soud(7, 3, k)
          |             fun_front_up(adresse_bp_cobot)
          |             tab_arc_ret_g[k] =  get_actual_tcp_pose() 	    #Enregistrer position dans tableau retrait quand appui Bp_cobot
          |             close_popup()
          |             end_teach_mode()
          |             global reglage_g = 0
          | 
          |             sync()
          | 
          |         ##############################################################################
          | 
          |     ##############################################################################
          | 
          | ############################soudure cercle####################################
          | 
          |     #################################################################################
          | 
          |         elif reglage_g == 4:                                  #remplissage tableau
          |             teach_mode()
          |             fun_popup_soud(1, 4, l)
          |             fun_front_up(adresse_bp_cobot)
          |             tab_cer_app_g[l] =  get_actual_tcp_pose()     	#Enregistrer position dans tableau d approche des soudures arc de cercle quand appui Bp_cobot
          |             close_popup()
          | 
          |             fun_popup_soud(2, 4, l)
          |             fun_front_up(adresse_bp_cobot)
          |             tab_cer_deb_g[l] =  get_actual_tcp_pose()     	#Enregistrer position dans tableau debut quand appui Bp_cobot
          |             close_popup()
          | 
          |             fun_popup_soud(3, 4, l)
          |             fun_front_up(adresse_bp_cobot)
          |             tab_cer_quart_g[l] =  get_actual_tcp_pose()   	#Enregistrer position dans tableau d'approche des soudures arc de cercle quand appui Bp_cobot
          |             close_popup()
          | 
          |             fun_popup_soud(4, 4, l)
          |             fun_front_up(adresse_bp_cobot)
          |             tab_cer_mil_g[l] =  get_actual_tcp_pose()     	#Enregistrer position dans tableau milieu quand appui Bp_cobot
          |             close_popup()
          | 
          |             fun_popup_soud(5, 4, l)
          |             fun_front_up(adresse_bp_cobot)
          |             tab_cer_tro_g[l] =  get_actual_tcp_pose()     	#Enregistrer position dans tableau milieu quand appui Bp_cobot
          |             close_popup()
          | 
          |             fun_popup_soud(6, 4, l)
          |             fun_front_up(adresse_bp_cobot)
          |             tab_cer_fin_g[l] =  get_actual_tcp_pose()     	#Enregistrer position dans un tableau fin quand appui Bp_cobot
          |             close_popup()
          | 
          |             vit_cer_g[l] = fun_demande_vit(4)
          | 
          |             fun_popup_soud(7, 4, l)
          |             fun_front_up(adresse_bp_cobot)
          |             tab_cer_ret_g[l] =  get_actual_tcp_pose()    	#position de retrait est la meme que position d approche
          |             close_popup()
          |             end_teach_mode()
          |             global reglage_g = 0
          |             sync()
          | 
          |         end
          | 
          |     ##############################################################################
          | 
          | ############################################################
        Script: sync()
      Script: sync()
    Script: sync()
Thread Thread_10 (runOnlyOnce=false)
  Folder reglage [hidden by the author, left out]
  Script: sync()
